// TIA Portal V19 export
FUNCTION_BLOCK "Alarms"   // FB7, LAD
{ S7_Optimized_Access := 'TRUE' }
// stored: MemoryReserve 100, SetENOAutomatically false
   VAR_TEMP   // added for the SCL form of the ladder/FBD networks
      _w1 : Bool;
      _w2 : Bool;
      _w3 : Bool;
   END_VAR
BEGIN

REGION Network 1: IBC Valve Open Fault
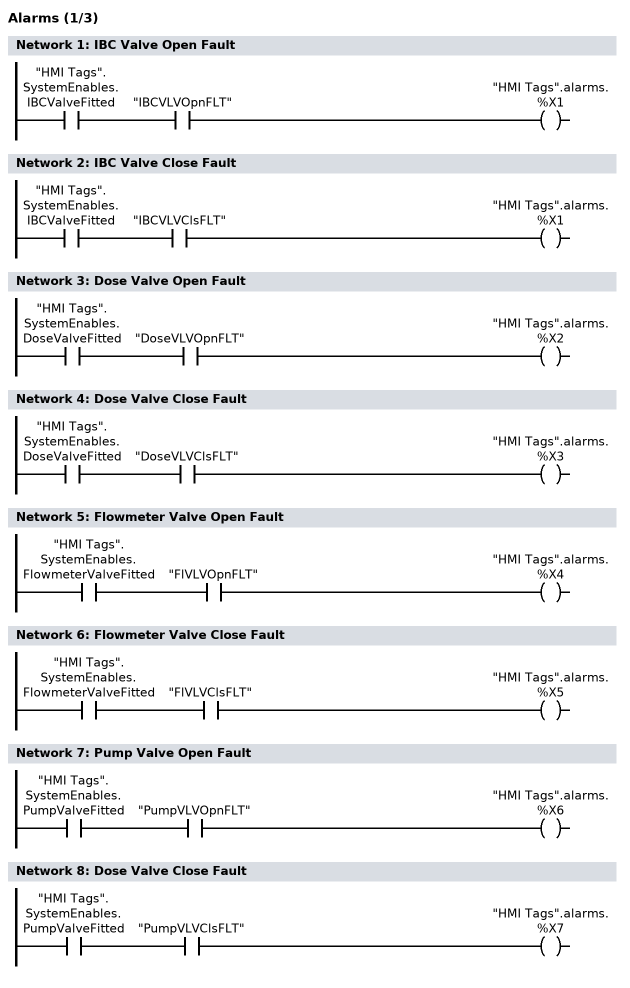
   RUNG wire#powerrail
      Contact( "HMI Tags".SystemEnables.IBCValveFitted )
      Contact( "IBCVLVOpnFLT" )
      Coil( "HMI Tags".alarms.%X1 )
   END_RUNG
   // the same network as SCL:
   "HMI Tags".alarms.%X1 := "HMI Tags".SystemEnables.IBCValveFitted AND "IBCVLVOpnFLT";
END_REGION

REGION Network 2: IBC Valve Close Fault
   RUNG wire#powerrail
      Contact( "HMI Tags".SystemEnables.IBCValveFitted )
      Contact( "IBCVLVClsFLT" )
      Coil( "HMI Tags".alarms.%X1 )
   END_RUNG
   // the same network as SCL:
   "HMI Tags".alarms.%X1 := "HMI Tags".SystemEnables.IBCValveFitted AND "IBCVLVClsFLT";
END_REGION

REGION Network 3: Dose Valve Open Fault
   RUNG wire#powerrail
      Contact( "HMI Tags".SystemEnables.DoseValveFitted )
      Contact( "DoseVLVOpnFLT" )
      Coil( "HMI Tags".alarms.%X2 )
   END_RUNG
   // the same network as SCL:
   "HMI Tags".alarms.%X2 := "HMI Tags".SystemEnables.DoseValveFitted AND "DoseVLVOpnFLT";
END_REGION

REGION Network 4: Dose Valve Close Fault
   RUNG wire#powerrail
      Contact( "HMI Tags".SystemEnables.DoseValveFitted )
      Contact( "DoseVLVClsFLT" )
      Coil( "HMI Tags".alarms.%X3 )
   END_RUNG
   // the same network as SCL:
   "HMI Tags".alarms.%X3 := "HMI Tags".SystemEnables.DoseValveFitted AND "DoseVLVClsFLT";
END_REGION

REGION Network 5: Flowmeter Valve Open Fault
   RUNG wire#powerrail
      Contact( "HMI Tags".SystemEnables.FlowmeterValveFitted )
      Contact( "FlVLVOpnFLT" )
      Coil( "HMI Tags".alarms.%X4 )
   END_RUNG
   // the same network as SCL:
   "HMI Tags".alarms.%X4 := "HMI Tags".SystemEnables.FlowmeterValveFitted AND "FlVLVOpnFLT";
END_REGION

REGION Network 6: Flowmeter Valve Close Fault
   RUNG wire#powerrail
      Contact( "HMI Tags".SystemEnables.FlowmeterValveFitted )
      Contact( "FlVLVClsFLT" )
      Coil( "HMI Tags".alarms.%X5 )
   END_RUNG
   // the same network as SCL:
   "HMI Tags".alarms.%X5 := "HMI Tags".SystemEnables.FlowmeterValveFitted AND "FlVLVClsFLT";
END_REGION

REGION Network 7: Pump Valve Open Fault
   RUNG wire#powerrail
      Contact( "HMI Tags".SystemEnables.PumpValveFitted )
      Contact( "PumpVLVOpnFLT" )
      Coil( "HMI Tags".alarms.%X6 )
   END_RUNG
   // the same network as SCL:
   "HMI Tags".alarms.%X6 := "HMI Tags".SystemEnables.PumpValveFitted AND "PumpVLVOpnFLT";
END_REGION

REGION Network 8: Dose Valve Close Fault
   RUNG wire#powerrail
      Contact( "HMI Tags".SystemEnables.PumpValveFitted )
      Contact( "PumpVLVClsFLT" )
      Coil( "HMI Tags".alarms.%X7 )
   END_RUNG
   // the same network as SCL:
   "HMI Tags".alarms.%X7 := "HMI Tags".SystemEnables.PumpValveFitted AND "PumpVLVClsFLT";
END_REGION

REGION Network 9: Flowmeter not counting when required
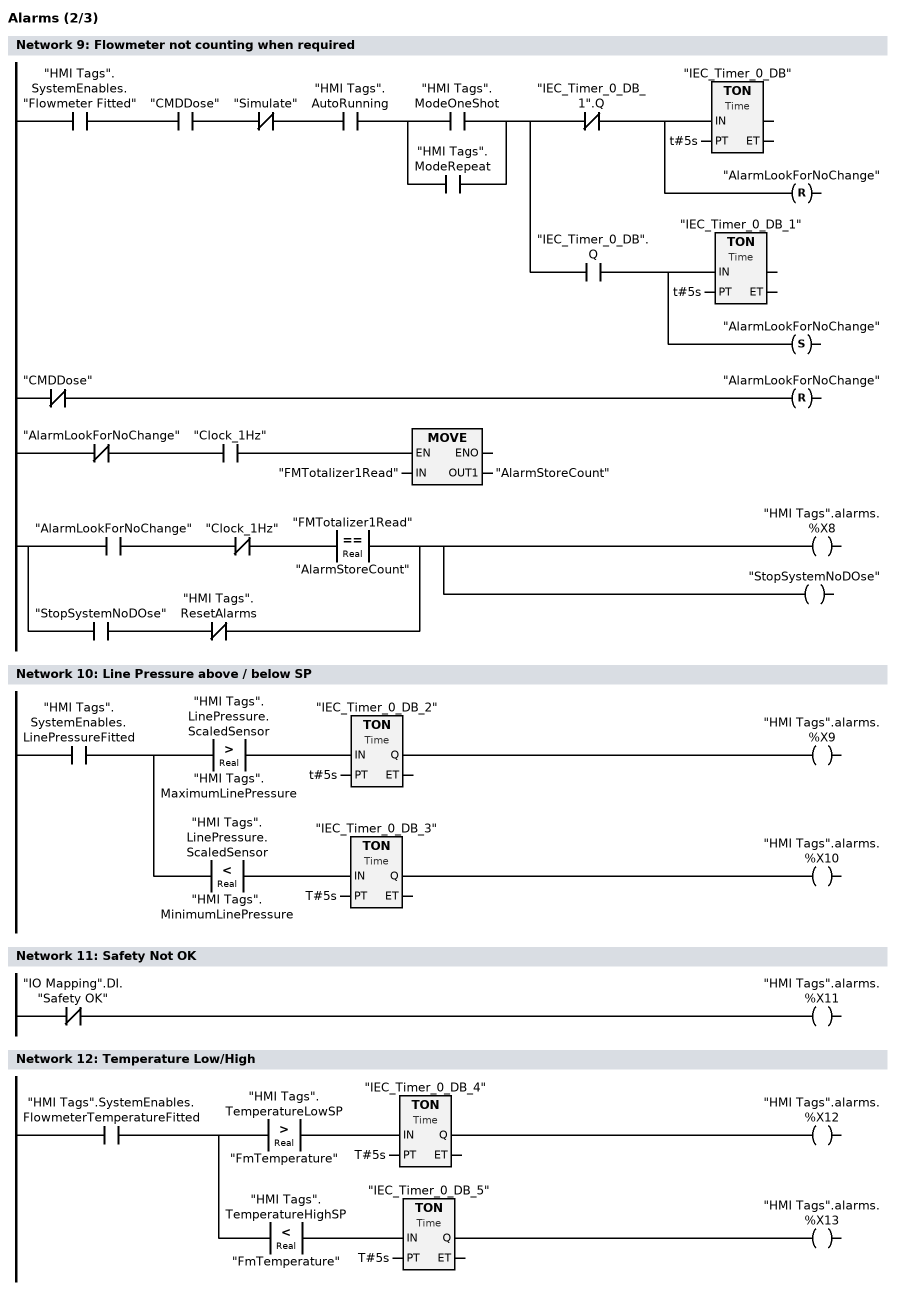
   RUNG wire#powerrail
      Contact( "HMI Tags".SystemEnables."Flowmeter Fitted" )
      Contact( "CMDDose" )
      I_Contact( "Simulate" )
      Contact( "HMI Tags".AutoRunning )
      wire#w1
      Contact( "HMI Tags".ModeOneShot )
      wire#w2
      I_Contact( "IEC_Timer_0_DB_1".Q )
      wire#w3
      { S7_Templates := "time_type := Time" } "IEC_Timer_0_DB".TON(pt := t#5s, et =>)
   END_RUNG
   RUNG wire#w1
      Contact( "HMI Tags".ModeRepeat )
   END_RUNG wire#w2
   RUNG wire#w3
      R_Coil( "AlarmLookForNoChange" )
   END_RUNG
   RUNG wire#w2
      Contact( "IEC_Timer_0_DB".Q )
      wire#w4
      { S7_Templates := "time_type := Time" } "IEC_Timer_0_DB_1".TON(pt := t#5s, et =>)
   END_RUNG
   RUNG wire#w4
      S_Coil( "AlarmLookForNoChange" )
   END_RUNG
   RUNG wire#powerrail
      I_Contact( "CMDDose" )
      R_Coil( "AlarmLookForNoChange" )
   END_RUNG
   RUNG wire#powerrail
      I_Contact( "AlarmLookForNoChange" )
      Contact( "Clock_1Hz" )
      Move(in := "FMTotalizer1Read", out1 => "AlarmStoreCount")
   END_RUNG
   RUNG wire#powerrail
      Contact( "AlarmLookForNoChange" )
      I_Contact( "Clock_1Hz" )
      { S7_Templates := "SrcType := Real" } EQ_Contact(in1 := "FMTotalizer1Read", in2 := "AlarmStoreCount")
      wire#w5
      Coil( "HMI Tags".alarms.%X8 )
   END_RUNG
   RUNG wire#powerrail
      Contact( "StopSystemNoDOse" )
      I_Contact( "HMI Tags".ResetAlarms )
   END_RUNG wire#w5
   RUNG wire#w5
      Coil( "StopSystemNoDOse" )
   END_RUNG
   // the same network as SCL:
   #_w1 := "HMI Tags".SystemEnables."Flowmeter Fitted" AND "CMDDose" AND NOT "Simulate" AND "HMI Tags".AutoRunning AND ("HMI Tags".ModeOneShot OR "HMI Tags".ModeRepeat);
   #_w2 := #_w1 AND NOT "IEC_Timer_0_DB_1".Q;
   "IEC_Timer_0_DB".TON(IN := #_w2, PT := t#5s);
   IF #_w2 THEN "AlarmLookForNoChange" := FALSE; END_IF;
   #_w3 := #_w1 AND "IEC_Timer_0_DB".Q;
   "IEC_Timer_0_DB_1".TON(IN := #_w3, PT := t#5s);
   IF #_w3 THEN "AlarmLookForNoChange" := TRUE; END_IF;
   IF NOT "CMDDose" THEN "AlarmLookForNoChange" := FALSE; END_IF;
   IF NOT "AlarmLookForNoChange" AND "Clock_1Hz" THEN "AlarmStoreCount" := "FMTotalizer1Read"; END_IF;
   "HMI Tags".alarms.%X8 := ("AlarmLookForNoChange" AND NOT "Clock_1Hz" AND ("FMTotalizer1Read" = "AlarmStoreCount")) OR ("StopSystemNoDOse" AND NOT "HMI Tags".ResetAlarms);
   "StopSystemNoDOse" := "HMI Tags".alarms.%X8;
END_REGION

REGION Network 10: Line Pressure above / below SP
   RUNG wire#powerrail
      Contact( "HMI Tags".SystemEnables.LinePressureFitted )
      wire#w1
      { S7_Templates := "SrcType := Real" } GT_Contact(in1 := "HMI Tags".LinePressure.ScaledSensor, in2 := "HMI Tags".MaximumLinePressure)
      { S7_Templates := "time_type := Time" } "IEC_Timer_0_DB_2".TON(pt := t#5s, et =>)
      Coil( "HMI Tags".alarms.%X9 )
   END_RUNG
   RUNG wire#w1
      { S7_Templates := "SrcType := Real" } LT_Contact(in1 := "HMI Tags".LinePressure.ScaledSensor, in2 := "HMI Tags".MinimumLinePressure)
      { S7_Templates := "time_type := Time" } "IEC_Timer_0_DB_3".TON(pt := T#5s, et =>)
      Coil( "HMI Tags".alarms.%X10 )
   END_RUNG
   // the same network as SCL:
   "IEC_Timer_0_DB_2".TON(IN := "HMI Tags".SystemEnables.LinePressureFitted AND ("HMI Tags".LinePressure.ScaledSensor > "HMI Tags".MaximumLinePressure),
                          PT := t#5s);
   "HMI Tags".alarms.%X9 := "IEC_Timer_0_DB_2".Q;
   "IEC_Timer_0_DB_3".TON(IN := "HMI Tags".SystemEnables.LinePressureFitted AND ("HMI Tags".LinePressure.ScaledSensor < "HMI Tags".MinimumLinePressure),
                          PT := T#5s);
   "HMI Tags".alarms.%X10 := "IEC_Timer_0_DB_3".Q;
END_REGION

REGION Network 11: Safety Not OK
   RUNG wire#powerrail
      I_Contact( "IO Mapping".DI."Safety OK" )
      Coil( "HMI Tags".alarms.%X11 )
   END_RUNG
   // the same network as SCL:
   "HMI Tags".alarms.%X11 := NOT "IO Mapping".DI."Safety OK";
END_REGION

REGION Network 12: Temperature Low/High
   RUNG wire#powerrail
      Contact( "HMI Tags".SystemEnables.FlowmeterTemperatureFitted )
      wire#w1
      { S7_Templates := "SrcType := Real" } GT_Contact(in1 := "HMI Tags".TemperatureLowSP, in2 := "FmTemperature")
      { S7_Templates := "time_type := Time" } "IEC_Timer_0_DB_4".TON(pt := T#5s, et =>)
      Coil( "HMI Tags".alarms.%X12 )
   END_RUNG
   RUNG wire#w1
      { S7_Templates := "SrcType := Real" } LT_Contact(in1 := "HMI Tags".TemperatureHighSP, in2 := "FmTemperature")
      { S7_Templates := "time_type := Time" } "IEC_Timer_0_DB_5".TON(pt := T#5s, et =>)
      Coil( "HMI Tags".alarms.%X13 )
   END_RUNG
   // the same network as SCL:
   "IEC_Timer_0_DB_4".TON(IN := "HMI Tags".SystemEnables.FlowmeterTemperatureFitted AND ("HMI Tags".TemperatureLowSP > "FmTemperature"),
                          PT := T#5s);
   "HMI Tags".alarms.%X12 := "IEC_Timer_0_DB_4".Q;
   "IEC_Timer_0_DB_5".TON(IN := "HMI Tags".SystemEnables.FlowmeterTemperatureFitted AND ("HMI Tags".TemperatureHighSP < "FmTemperature"),
                          PT := T#5s);
   "HMI Tags".alarms.%X13 := "IEC_Timer_0_DB_5".Q;
END_REGION

REGION Network 13: VFDFAULT
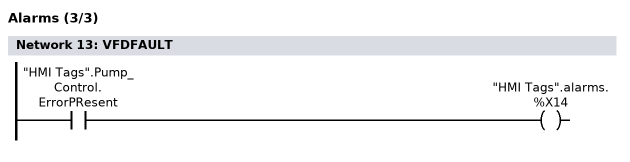
   RUNG wire#powerrail
      Contact( "HMI Tags".Pump_Control.ErrorPResent )
      Coil( "HMI Tags".alarms.%X14 )
   END_RUNG
   // the same network as SCL:
   "HMI Tags".alarms.%X14 := "HMI Tags".Pump_Control.ErrorPResent;
END_REGION
END_FUNCTION_BLOCK
